Yaskawa INFORM job: OUT1.JBI

/JOB
//NAME OUT1
//POS
///NPOS 0,0,0,0,0,0
//INST
///DATE 2018/06/13 13:49
///ATTR SC,RW
NOP
DOUT OT#(1) ON
DOUT OT#(2) ON
DOUT OT#(3) ON
END
